INTERFACE I_Visitor

METHOD visitConveyor
VAR_INPUT
	fbConveyor : FB_Conveyor;
END_VAR
END_METHOD

METHOD visitHeater
VAR_INPUT
	fbHeater : FB_Heater;
END_VAR
END_METHOD

METHOD visitIPC
VAR_INPUT
	fbIPC : FB_IPCDiagnostics;
END_VAR
END_METHOD

END_INTERFACE

(* stored: Version 1.1.0.1, ProductVersion 3.1.4024.12
   Itf I_Visitor: Id {ca293700-6744-4e91-b2aa-c10eff183998}
   Method visitConveyor: Id {674d8e4c-61e3-4817-b84b-3ea9ba4e51d1}
   Method visitHeater: Id {3c75bc6f-c2b0-4f18-aa1e-655777d0dd14}
   Method visitIPC: Id {85bdd0c6-6121-41ee-a678-4ee8c40079f0} *)
